SUBAPPLICATION Uebung_026 (* Spiegelabfolge (6) *)
  (* Standard: 61499-2; Description: Copyright (c) 2023 Meisterschulen am Ostbahnhof This program and the accompanying materials are made available under the terms of the Eclipse Public License 2.0 which is available at https://www.eclipse.org/legal/epl-2.0/ SPDX-License-Identifier: EPL-2.0 *)
  (* Version 1.0, 2023-10-23, Franz Höpfinger, Meisterschulen am Ostbahnhof, initial API and implementation and/or initial documentation *)
  PACKAGE Uebungen;
  IMPORT isobus::UT::io::Softkey::SoftKeyActivationCode::SK_PRESSED;
  IMPORT isobus::UT::io::Softkey::SoftKeyActivationCode::SK_RELEASED;
  IMPORT Uebungen::const::UT::DefaultPool::SoftKey_F1;
  IMPORT Uebungen::const::UT::DefaultPool::SoftKey_F2;
  IMPORT Uebungen::const::UT::DefaultPool::SoftKey_F3;
  IMPORT Uebungen::const::UT::DefaultPool::SoftKey_F8;
  IMPORT Uebungen::const::UT::DefaultPool::SoftKey_F9;
  IMPORT logiBUS::io::DQ::logiBUS_DO::Output_Q1;
  IMPORT logiBUS::io::DQ::logiBUS_DO::Output_Q2;
  IMPORT logiBUS::io::DQ::logiBUS_DO::Output_Q3;
  IMPORT logiBUS::io::DQ::logiBUS_DO::Output_Q4;
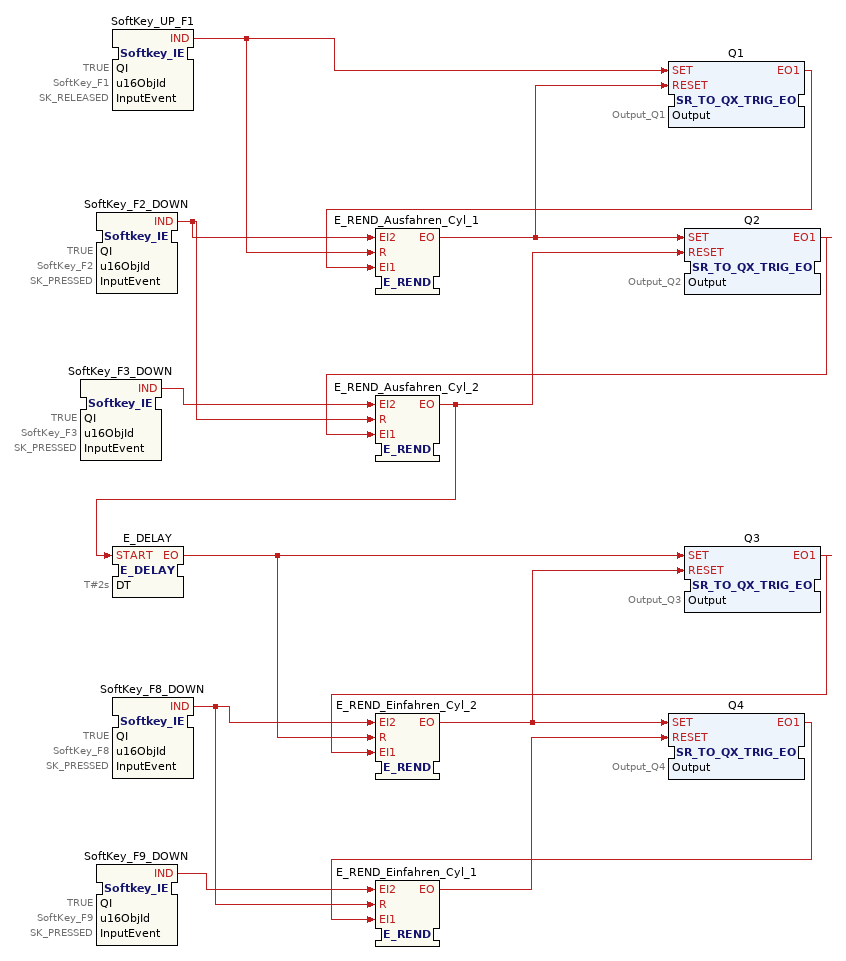
  (* START-Knopf Ausfahren *)
  (* Endlage Ausfahren_Cyl_1 *)
  (* Endlage Ausfahren_Cyl_2 *)
  (* Ausfahren_Cyl_1 *)
  (* Ausfahren_Cyl_2 *)
  (* Einfahren Zeit gesteuert *)
  (* Endlage Einfahren_Cyl_1 *)
  (* Einfahren_Cyl_2 *)
  (* Endlage Einfahren_Cyl_2 *)
  (* Einfahren_Cyl_1 *)
  FBS
    SoftKey_UP_F1 : isobus::UT::io::Softkey::Softkey_IE(QI := TRUE, u16ObjId := SoftKey_F1, InputEvent := SK_RELEASED);
    SoftKey_F2_DOWN : isobus::UT::io::Softkey::Softkey_IE(QI := TRUE, u16ObjId := SoftKey_F2, InputEvent := SK_PRESSED);
    SoftKey_F3_DOWN : isobus::UT::io::Softkey::Softkey_IE(QI := TRUE, u16ObjId := SoftKey_F3, InputEvent := SK_PRESSED);
    SoftKey_F9_DOWN : isobus::UT::io::Softkey::Softkey_IE(QI := TRUE, u16ObjId := SoftKey_F9, InputEvent := SK_PRESSED);
    SoftKey_F8_DOWN : isobus::UT::io::Softkey::Softkey_IE(QI := TRUE, u16ObjId := SoftKey_F8, InputEvent := SK_PRESSED);
    E_DELAY : iec61499::events::E_DELAY(DT := T#2s);
    E_REND_Ausfahren_Cyl_1 : iec61499::events::E_REND;
    E_REND_Ausfahren_Cyl_2 : iec61499::events::E_REND;
    E_REND_Einfahren_Cyl_2 : iec61499::events::E_REND;
    E_REND_Einfahren_Cyl_1 : iec61499::events::E_REND;
  END_FBS
  SUBAPPS
    Q4 : MyLib::sys::SR_TO_QX_TRIG_EO(Output := Output_Q4);
    Q2 : MyLib::sys::SR_TO_QX_TRIG_EO(Output := Output_Q2);
    Q3 : MyLib::sys::SR_TO_QX_TRIG_EO(Output := Output_Q3);
    Q1 : MyLib::sys::SR_TO_QX_TRIG_EO(Output := Output_Q1);
  END_SUBAPPS
  EVENT_CONNECTIONS
    SoftKey_F2_DOWN.IND TO E_REND_Ausfahren_Cyl_1.EI2;
    SoftKey_F3_DOWN.IND TO E_REND_Ausfahren_Cyl_2.EI2;
    SoftKey_F9_DOWN.IND TO E_REND_Einfahren_Cyl_1.EI2;
    SoftKey_F8_DOWN.IND TO E_REND_Einfahren_Cyl_2.EI2;
    E_REND_Ausfahren_Cyl_2.EO TO E_DELAY.START;
    SoftKey_UP_F1.IND TO E_REND_Ausfahren_Cyl_1.R;
    SoftKey_F2_DOWN.IND TO E_REND_Ausfahren_Cyl_2.R;
    E_DELAY.EO TO E_REND_Einfahren_Cyl_2.R;
    SoftKey_F8_DOWN.IND TO E_REND_Einfahren_Cyl_1.R;
    E_REND_Einfahren_Cyl_2.EO TO Q4.SET;
    E_REND_Einfahren_Cyl_1.EO TO Q4.RESET;
    Q4.EO1 TO E_REND_Einfahren_Cyl_1.EI1;
    E_REND_Ausfahren_Cyl_1.EO TO Q2.SET;
    E_REND_Ausfahren_Cyl_2.EO TO Q2.RESET;
    Q2.EO1 TO E_REND_Ausfahren_Cyl_2.EI1;
    E_DELAY.EO TO Q3.SET;
    E_REND_Einfahren_Cyl_2.EO TO Q3.RESET;
    Q3.EO1 TO E_REND_Einfahren_Cyl_2.EI1;
    SoftKey_UP_F1.IND TO Q1.SET;
    E_REND_Ausfahren_Cyl_1.EO TO Q1.RESET;
    Q1.EO1 TO E_REND_Ausfahren_Cyl_1.EI1;
  END_CONNECTIONS
END_SUBAPPLICATION
